(* CODESYS project gittest

Project tree, tasks and I/O mapping:
  Device : 750-8210 PFC200, WAGO, order no. 750-8210, version 6.0.0.15
    application Application
      libraries: Standard, * (System)
      task MainTask (cyclic, interval t#50ms, priority 15) calls PLC_PRG
      program PLC_PRG [ST]
    Kbus : Kbus, WAGO, version 2.1.0.1
        unmapped channels: K-BUS diagnostics
*)

// Device/Application/PLC_PRG
PROGRAM PLC_PRG
VAR
	a: INT;
END_VAR

a := a+1;

END_PROGRAM
